PROGRAM OP140_Error
VAR
	Step_No: INT;
	AutoStepErr_1: TON;
	OP140_StepErr1: TON;
	OP140_StepErr2: TON;
END_VAR

// Set ERROR ACTIVE
IF ((OP140_ErrorWord_0= 1) OR (OP140_ErrorWord_1= 1) OR (OP140_ErrorWord_2= 1)) THEN
	OP140_ErrorActive:= TRUE;
	END_IF
	//Reset ErrorActive
IF (OP140_HMI_Reset) THEN 
	OP140_ErrorActive:= FALSE;
	OP140_ErrorWord_0:= 0;
	OP140_ErrorWord_1:= 0;
	Op140_ErrorWord_2:= 0;
	END_IF
	
//Step Errors


IF OP140_AutoSequence.OP140_Leak_Test_1.Step_No=40 AND  NOT OP140_AutoSequence.OP140_Leak_Test_1.Axis_In_Pos AND OP140_StepErr1.q THEN
OP140_ErrorWord_0.0:=TRUE;
END_IF
IF OP140_AutoSequence.OP140_Leak_Test_1.Step_No=80 AND  NOT OP140_AutoSequence.OP140_Leak_Test_1.Axis_In_home AND OP140_StepErr2.q THEN
OP140_ErrorWord_0.1:=TRUE;
END_IF
IF OP140_AutoSequence.OP140_Leak_Test_1.LH_ATEQ_FB.Result_Error=TRUE THEN
	OP140_ErrorWord_0.2:=TRUE;
	
END_IF
IF OP140_AutoSequence.OP140_Leak_Test_1.RH_ATEQ_FB.Result_Error=TRUE THEN
	OP140_ErrorWord_0.3:=TRUE;
	
END_IF


	OP140_StepErr1(IN:=OP140_AutoSequence.OP140_Leak_Test_1.Step_No=40 , PT:=T#2S , Q=> , ET=> );
	OP140_StepErr2(IN:=OP140_AutoSequence.OP140_Leak_Test_1.Step_No=80 , PT:=T#2S , Q=> , ET=> );

END_PROGRAM

(* stored: Version 1.1.0.1, ProductVersion 3.1.4024.11
   POU OP140_Error: Id {ac65b6e6-27bf-4de3-9923-224b69f44c75}, SpecialFunc None *)
